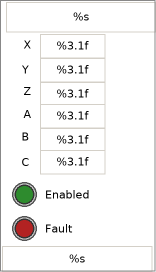
VISUALIZATION V_Mover  // 156x272
VAR_IN_OUT
	Mover : ST_Mover_HMI;
	Position : Position6D;
END_VAR
    Label (14,30 27x30), "X"
    Label (12,58 27x24), "Y"
    Label (14,80 27x23), "Z"
    Label (14,104 27x21), "A"
    Label (12,124 27x26), "B"
    Label (12,152 27x21), "C"
    Textfield (40,34 65x24), "%3.1f", text variable: Position.x
    Textfield (40,58 65x24), "%3.1f", text variable: Position.y
    Textfield (40,82 65x24), "%3.1f", text variable: Position.z
    Textfield (40,104 65x24), "%3.1f", text variable: Position.a
    Textfield (40,128 65x24), "%3.1f", text variable: Position.b
    Textfield (40,150 65x24), "%3.1f", text variable: Position.c
    Lamp1 (10,180 29x29), variable: Mover.Status.Enabled, style: Lamp-Lamp1-Green
    Label (42,182 107x26), "Enabled"
    Textfield (6,2 150x30), "%s", text variable: Mover.Status.ID
    Textfield (2,246 150x26), "%s", text variable: Mover.Status.CommandMode
    Lamp1 (10,214 29x29), variable: Mover.Status.Error, style: Lamp-Lamp1-Red
    Label (42,216 107x26), "Fault"
END_VISUALIZATION

(* stored: Version 1.1.0.1, ProductVersion 3.1.4024.12
   Visu V_Mover: Id {507c57e0-0a29-487b-ac40-679445be6fa1} *)
